FUNCTION_BLOCK FB_ReadCoilExample
VAR
	fbMBReadCoils : FB_MBReadCoils;
	nReadValue : BYTE;
	aStateMachine : (WAIT, TRIGGER, READ);
	fbTrigger : R_TRIG;
END_VAR

fbTrigger();
IF fbTrigger.Q THEN
	IF aStateMachine := WAIT THEN
		aStateMachine := TRIGGER;
	END_IF
END_IF
CASE aStateMachine OF
	WAIT:
		// do nothing
	TRIGGER:
		fbMBReadCoils(
		sIPAddr:= '192.168.5.34' , // IP of virtual machine
		nTCPPort:= , 
		nUnitID:= , 
		nQuantity:= , 
		nMBAddr:= , 
		cbLength:= SIZEOF(nReadValue), 
		pDestAddr:= ADR(nReadValue), 
		bExecute:= TRUE, 
		tTimeout:= , 
		bBusy=> , 
		bError=> , 
		nErrId=> , 
		cbRead=> );
		
		aStateMachine := READ;
	READ:
		// waite for response
		fbMBReadCoils(bExecute := FALSE); // read until we get sth from modbus app in windows
		IF NOT fbMBReadCoils.bBusy OR fbMBReadCoils.bError THEN
			aStateMachine := WAIT;
		END_IF
	
END_CASE

END_FUNCTION_BLOCK

(* stored: Version 1.1.0.1, ProductVersion 3.1.4024.12
   POU FB_ReadCoilExample: Id {67787ba6-a0c7-477e-9f3e-97f287d04096}, SpecialFunc None *)
